TYPE
    ST_DoubleValve EXTENDS ST_SignleValve :
    STRUCT
        Retract : BOOL;
    END_STRUCT
END_TYPE

(* stored: Version 1.1.0.1, ProductVersion 3.1.4024.13
   DUT ST_DoubleValve: Id {70e2fc7d-dc20-4355-a6de-e763b1550ab2} *)
